{attribute 'enable_dynamic_creation'}
FUNCTION_BLOCK FB_TaskMoveToPosition EXTENDS FB_AbstructFuture
VAR_OUTPUT
END_VAR
VAR
	_v				: MC_LREAL;
	_a				: MC_LREAL;
	_d				: MC_LREAL;
	_j				: MC_LREAL;
	_pos_x 			: LREAL;
	_pos_y 			: LREAL;
	_pos_c			: LREAL;
	_dynamics		: DynamicConstraint_PathXY;
	_position 		: PositionXYC;
	_error_id		: UDINT;
	_mover		: REFERENCE TO MC_PlanarMover;
	_cmdFB			: MC_PlanarFeedback;
	_prohibit 		: BOOL;
	_abort_executor : FB_Executor;
	_state_num 			:UINT;
	_abort_state	:UINT;
END_VAR

{warning 'add method implementation '}
METHOD abort : BOOL
_cmdFB.Update();
_state_num := 0;
CASE _abort_state OF
	0:
		IF _cmdFB.Active THEN
			_dynamics.SetValuesVADJ(2000,20000,200000,200000);
			_abort_state := 1;
		ELSE
			abort := TRUE;
		END_IF
	1:
		//停止
		_mover.Halt(_cmdFB,_dynamics);
		_abort_state := 2;
	2:
		//停止完了フラグ待ち
		IF _cmdFB.Done THEN
			abort := TRUE;
			_error_id := 0;
		END_IF
		IF _cmdFB.Error THEN
			abort := TRUE;
			_error_id := _cmdFB.ErrorId;
		END_IF
END_CASE
END_METHOD

{warning 'add method implementation '}
METHOD execute : BOOL
_cmdFB.Update();
_abort_state := 0;
CASE _state_num OF
	0:
		//直線運動
		IF NOT _cmdFB.Active AND NOT _cmdFB.Busy THEN
			_mover.MoveToPosition(_cmdFB,_position,_dynamics,0);
			_state_num := 1;
		END_IF
	1:
		//直線運動の完了フラグ待ち
		IF _cmdFB.Done THEN
			execute := TRUE;
			_error_id := 0;
		END_IF
		IF _cmdFB.Error THEN
			execute := TRUE;
			_error_id := _cmdFB.ErrorId;
		END_IF
END_CASE
END_METHOD

{warning 'add method implementation '}
METHOD init : BOOL
IF _prohibit THEN
	_error_id := 16#80000000;
	init := TRUE;
ELSIF _v = 0 OR _a = 0 OR _d = 0 THEN
	_error_id := 1;
	init := TRUE;
ELSE
	_dynamics.SetValuesVADJ(_v, _a, _d, _j);
	_position.SetValuesXYC(_pos_x, _pos_y, _pos_c);
	_abort_executor.init();
	_error_id := 0;
	_state_num := 0;
	_abort_state := 0;
	init := TRUE;
END_IF
END_METHOD

PROPERTY mover : REFERENCE TO MC_PlanarMover
SET
_mover REF= mover;
END_SET
END_PROPERTY

{warning 'add property implementation'}
PROPERTY nErrorID : UDINT
GET
nErrorID := _error_id;
END_GET
END_PROPERTY

{warning 'add method implementation '}
METHOD quit : BOOL
init();
quit := TRUE;
END_METHOD

METHOD set_dynamics : BOOL
VAR_INPUT
	v: MC_LREAL;
	a: MC_LREAL;
	d: MC_LREAL;
	j: MC_LREAL;
END_VAR
_v := v;
_a := a;
_d := d;
_j := j;
set_dynamics := TRUE;
END_METHOD

METHOD set_target_position : BOOL
VAR_INPUT
	x: LREAL;
	y: LREAL;
	c: LREAL;
END_VAR
_pos_x := x;
_pos_y := y;
_pos_c := c;

set_target_position := TRUE;
END_METHOD

END_FUNCTION_BLOCK

(* stored: Version 1.1.0.1, ProductVersion 3.1.4024.12
   POU FB_TaskMoveToPosition: Id {2ec2db54-2fd0-4ec5-8d5f-0acb3a1d1c71}, SpecialFunc None
   Method abort: Id {ae2a45bb-2c60-4ac4-9b8e-2c704438498e}
   Method execute: Id {5269bf3b-d3fe-4a29-9d10-efacd53a1e73}
   Method init: Id {a571328b-641b-403a-992b-bae876238a59}
   Property mover: Id {e3b35138-a063-4366-85ea-6786cef227b7}
   Set Set: Id {4a11cf61-5035-4693-b60e-058c96137679}
   Property nErrorID: Id {a5a03649-4296-4991-9d72-d5144728d1a2}
   Get Get: Id {445d43c2-7e42-451b-9bd7-8204f23f0250}
   Method quit: Id {fda1d651-d6bf-4840-8b98-1c5c46b6f2b3}
   Method set_dynamics: Id {f5e62bd7-bab2-4251-a23a-77e2c16f1e6b}
   Method set_target_position: Id {476622d5-869b-4d7f-9c13-ce8ef2b420a8} *)
